// TwinCAT 3 PLC project Radio
// ProgramVersion: 3.1.4024.0
// libraries:
//   Tc2_Standard, * (Beckhoff Automation GmbH)
//   Tc2_System, * (Beckhoff Automation GmbH)
//   Tc3_Module, * (Beckhoff Automation GmbH)
// project tree:
//   / PlcTask.TcTTO
//   POUs/ MAIN.TcPOU
// (motion and I/O tree: see PLC project trappenhuis_extraverlenging)
// real-time tasks:
//   TASK PlcTask: cycle T#10ms, priority 20, ADS port 350
//   TASK PlcTask1: cycle T#10ms, priority 21, ADS port 351
//   TASK PlcTask2: cycle T#10ms, priority 22, ADS port 352
//   TASK PlcTask3: cycle T#10ms, priority 23, ADS port 353
//   TASK PlcTask4: cycle T#10ms, priority 24, ADS port 354
//   TASK PlcTask5: cycle T#10ms, priority 25, ADS port 355
//   TASK PlcTask6: cycle T#10ms, priority 26, ADS port 356
//   TASK PlcTask7: cycle T#10ms, priority 27, ADS port 357
//   TASK PlcTask8: cycle T#10ms, priority 28, ADS port 358
//   TASK PlcTask9: cycle T#10ms, priority 29, ADS port 359
//   TASK PlcTask10: cycle T#10ms, priority 30, ADS port 360

CONFIGURATION Radio
    RESOURCE PLC ON TwinCAT3
        TASK PlcTask(INTERVAL := T#10ms, PRIORITY := 26);
        PROGRAM MAIN WITH PlcTask : MAIN;
    END_RESOURCE
END_CONFIGURATION

// ---- POUs/MAIN.TcPOU
PROGRAM MAIN
VAR
    bPlusButton, bMinusButton, bPlusPressed, bMinusPressed: BOOL;
    rVoltage: REAL := 0.0; // Start voltage
    fbPlusTimer, fbMinusTimer: TON;
END_VAR

(*

Radio (3 regels code)

Ontwerp de sturing van de frequentiekeuze van een autoradio d.m.v. 2 drukknoppen ( + en - )
zodat er een DC-spanning wordt geleverd tussen 0 en 10 V.
Met één enkele klik verhoogt of verlaagt men de DC-spanning met 100mV 
en met een druk langer dan 1seconde veranderd de spanning met 500mv per seconde.
*)

fbPlusTimer(IN:=bPlusButton, PT:=T#1S); IF NOT bPlusButton AND bPlusPressed THEN rVoltage := MIN(10.0, rVoltage + 0.1); bPlusPressed := FALSE; ELSIF bPlusButton AND NOT bPlusPressed THEN bPlusPressed := TRUE; END_IF; IF fbPlusTimer.Q THEN rVoltage := MIN(10.0, rVoltage + 0.5); fbPlusTimer.IN:=bPlusButton; END_IF;
fbMinusTimer(IN:=bMinusButton, PT:=T#1s); IF NOT bMinusButton AND bMinusPressed THEN rVoltage := MAX(0.0, rVoltage - 0.1); bMinusPressed := FALSE; ELSIF bMinusButton AND NOT bMinusPressed THEN bMinusPressed := TRUE; END_IF; IF fbMinusTimer.Q THEN rVoltage := MAX(0.0, rVoltage - 0.5); fbMinusTimer.IN:=bMinusButton; END_IF;

END_PROGRAM
